FUNCTION Atan2 : LREAL//输出角度范围为[-pi,pi]
VAR_INPUT
	y : LREAL;
	x : LREAL;
END_VAR
VAR
END_VAR

IF ABS(x)<1E-6 THEN
	IF y>=0 THEN
		Atan2 := pi/2;
	ELSE
		Atan2 := -pi/2;
	END_IF
ELSE
	IF x<0 AND y>=0 THEN
		Atan2 := ATAN(y/x) + pi;
	ELSIF x<0 AND y<0 THEN
		Atan2 := ATAN(y/x) - pi;
	ELSE
		Atan2 := ATAN(y/x);
	END_IF
END_IF

END_FUNCTION

(* stored: Version 1.1.0.1, ProductVersion 3.1.4024.2
   POU Atan2: Id {852dd33c-be8f-4b96-9343-0b250d365706}, SpecialFunc None *)
